# EPICS autosave request: CARSApp/Db/CARS_80_motor_positions.req
# FILE... CARS_80_motor_settings.req
file "CARS_motor_positions.req", P=$(P), M=m1
file "CARS_motor_positions.req", P=$(P), M=m2
file "CARS_motor_positions.req", P=$(P), M=m3
file "CARS_motor_positions.req", P=$(P), M=m4
file "CARS_motor_positions.req", P=$(P), M=m5
file "CARS_motor_positions.req", P=$(P), M=m6
file "CARS_motor_positions.req", P=$(P), M=m7
file "CARS_motor_positions.req", P=$(P), M=m8
file "CARS_motor_positions.req", P=$(P), M=m9
file "CARS_motor_positions.req", P=$(P), M=m10
file "CARS_motor_positions.req", P=$(P), M=m11
file "CARS_motor_positions.req", P=$(P), M=m12
file "CARS_motor_positions.req", P=$(P), M=m13
file "CARS_motor_positions.req", P=$(P), M=m14
file "CARS_motor_positions.req", P=$(P), M=m15
file "CARS_motor_positions.req", P=$(P), M=m16
file "CARS_motor_positions.req", P=$(P), M=m17
file "CARS_motor_positions.req", P=$(P), M=m18
file "CARS_motor_positions.req", P=$(P), M=m19
file "CARS_motor_positions.req", P=$(P), M=m20
file "CARS_motor_positions.req", P=$(P), M=m21
file "CARS_motor_positions.req", P=$(P), M=m22
file "CARS_motor_positions.req", P=$(P), M=m23
file "CARS_motor_positions.req", P=$(P), M=m24
file "CARS_motor_positions.req", P=$(P), M=m25
file "CARS_motor_positions.req", P=$(P), M=m26
file "CARS_motor_positions.req", P=$(P), M=m27
file "CARS_motor_positions.req", P=$(P), M=m28
file "CARS_motor_positions.req", P=$(P), M=m29
file "CARS_motor_positions.req", P=$(P), M=m30
file "CARS_motor_positions.req", P=$(P), M=m31
file "CARS_motor_positions.req", P=$(P), M=m32
file "CARS_motor_positions.req", P=$(P), M=m33
file "CARS_motor_positions.req", P=$(P), M=m34
file "CARS_motor_positions.req", P=$(P), M=m35
file "CARS_motor_positions.req", P=$(P), M=m36
file "CARS_motor_positions.req", P=$(P), M=m37
file "CARS_motor_positions.req", P=$(P), M=m38
file "CARS_motor_positions.req", P=$(P), M=m39
file "CARS_motor_positions.req", P=$(P), M=m40
file "CARS_motor_positions.req", P=$(P), M=m41
file "CARS_motor_positions.req", P=$(P), M=m42
file "CARS_motor_positions.req", P=$(P), M=m43
file "CARS_motor_positions.req", P=$(P), M=m44
file "CARS_motor_positions.req", P=$(P), M=m45
file "CARS_motor_positions.req", P=$(P), M=m46
file "CARS_motor_positions.req", P=$(P), M=m47
file "CARS_motor_positions.req", P=$(P), M=m48
file "CARS_motor_positions.req", P=$(P), M=m49
file "CARS_motor_positions.req", P=$(P), M=m50
file "CARS_motor_positions.req", P=$(P), M=m51
file "CARS_motor_positions.req", P=$(P), M=m52
file "CARS_motor_positions.req", P=$(P), M=m53
file "CARS_motor_positions.req", P=$(P), M=m54
file "CARS_motor_positions.req", P=$(P), M=m55
file "CARS_motor_positions.req", P=$(P), M=m56
file "CARS_motor_positions.req", P=$(P), M=m57
file "CARS_motor_positions.req", P=$(P), M=m58
file "CARS_motor_positions.req", P=$(P), M=m59
file "CARS_motor_positions.req", P=$(P), M=m60
file "CARS_motor_positions.req", P=$(P), M=m61
file "CARS_motor_positions.req", P=$(P), M=m62
file "CARS_motor_positions.req", P=$(P), M=m63
file "CARS_motor_positions.req", P=$(P), M=m64
file "CARS_motor_positions.req", P=$(P), M=m65
file "CARS_motor_positions.req", P=$(P), M=m66
file "CARS_motor_positions.req", P=$(P), M=m67
file "CARS_motor_positions.req", P=$(P), M=m68
file "CARS_motor_positions.req", P=$(P), M=m69
file "CARS_motor_positions.req", P=$(P), M=m70
file "CARS_motor_positions.req", P=$(P), M=m71
file "CARS_motor_positions.req", P=$(P), M=m72
file "CARS_motor_positions.req", P=$(P), M=m73
file "CARS_motor_positions.req", P=$(P), M=m74
file "CARS_motor_positions.req", P=$(P), M=m75
file "CARS_motor_positions.req", P=$(P), M=m76
file "CARS_motor_positions.req", P=$(P), M=m77
file "CARS_motor_positions.req", P=$(P), M=m78
file "CARS_motor_positions.req", P=$(P), M=m79
file "CARS_motor_positions.req", P=$(P), M=m80
